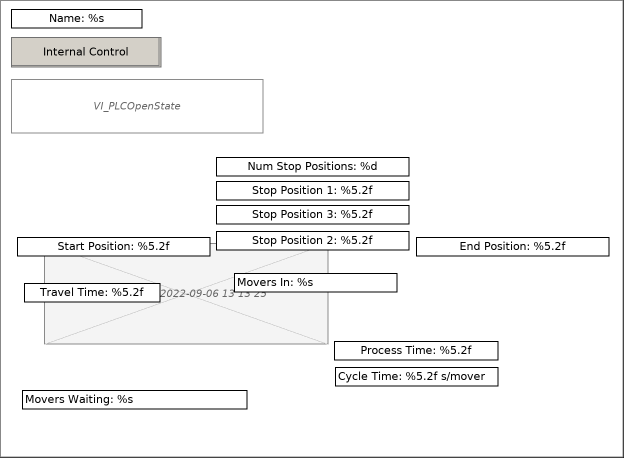
VISUALIZATION VI_StationVISU  // 624x458
VAR_IN_OUT
	fbStation : FB_Station;
END_VAR
    Rectangle (0,0 624x458)
    Frame (11,79 252x54)
        shows VI_PLCOpenState(bExecute := fbStation.bStart, sName := 'Secuence', bBusy := fbStation.stSecuenceStatus.bBusy, bDone := fbStation.stSecuenceStatus.bDone, bError := fbStation.stSecuenceStatus.bError, ErrorID := fbStation.stSecuenceStatus.udiErrorID)
    Button (11,37 150x30), "Internal Control", tooltip "Enable Visu Control, all methods will be locked"
        toggle fbStation.bInternalControl
    Rectangle (11,9 131x19), "Name: %s", text variable: fbStation.stCfg.sName
        OnMouseClick: write the text variable via Default
    Image (44,243 284x101), image: ImagePool.2022-09-06 13 13 25
    Rectangle (17,237 193x19), "Start Position: %5.2f", text variable: fbStation.stCfg.lrStartPosition
        OnMouseClick: write the text variable via Default
    Rectangle (416,237 193x19), "End Position: %5.2f", text variable: fbStation.stCfg.lrEndPosition
        OnMouseClick: write the text variable via Default
    Rectangle (234,273 163x19), "Movers In: %s", text variable: fbStation.sMoversIn
        OnMouseClick: write the text variable via Default
    Rectangle (22,390 225x19), "Movers Waiting: %s", text variable: fbStation.sMoversWaiting
        OnMouseClick: write the text variable via Default
    Rectangle (216,157 193x19), "Num Stop Positions: %d", text variable: fbStation.stCfg.uiNumStopPositions
        OnMouseClick: write the text variable via Default
    Rectangle (216,181 193x19), "Stop Position 1: %5.2f", text variable: fbStation.stCfg.lrStopPosition[1]
        OnMouseClick: write the text variable via Default
    Rectangle (216,231 193x19), "Stop Position 2: %5.2f", text variable: fbStation.stCfg.lrStopPosition[2], invisible if: fbStation.stCfg.uiNumStopPositions < 2
        OnMouseClick: write the text variable via Default
    Rectangle (216,205 193x19), "Stop Position 3: %5.2f", text variable: fbStation.stCfg.lrStopPosition[3], invisible if: fbStation.stCfg.uiNumStopPositions < 3
        OnMouseClick: write the text variable via Default
    Rectangle (335,367 163x19), "Cycle Time: %5.2f s/mover", text variable: (fbStation.lrActualProcessTime+fbStation.lrActualWaitingTime)/udint_to_lreal(fbStation.stCfg.uiNumStopPositions)
    Rectangle (24,283 136x19), "Travel Time: %5.2f", text variable: fbStation.stCfg.lrTravelTime
        OnMouseClick: write the text variable via Default
    Rectangle (334,341 164x19), "Process Time: %5.2f", text variable: fbStation.stCfg.lrProcessingTime
        OnMouseClick: write the text variable via Default
END_VISUALIZATION

(* stored: Version 1.1.0.1, ProductVersion 3.1.4024.11
   Visu VI_StationVISU: Id {de0729b5-f064-48c2-b489-33e37893a66b} *)
